TYPE TcoDatamanResults_v_5_x_x :
STRUCT
    Id : UINT;
    Code : UINT;
    Extended : UINT;
    Length : UINT;
    Data : ARRAY[0..TcoVisionParams.MAX_BYTE_ARRAY] OF BYTE;
END_STRUCT
END_TYPE

(* stored: Version 1.1.0.1, ProductVersion 3.1.4024.11
   DUT TcoDatamanResults_v_5_x_x: Id {beecb9b7-fd6e-0f66-0bfe-155d8e15fda4} *)
